PROGRAM F22_AggregationHandScanner
VAR

	fbBarcodeType					: FB_SYSTEM_BarcodeType;

	bPackBarcode					: BOOL;
	bOuterIntermediateBarcode		: BOOL;
	bOuterBarcode					: BOOL;
	bCaseBarcode					: BOOL;
	sPackBarcode					: T_PACK_Barcode;
	sOuterIntermediateBarcode		:  T_MaxString;
	sOuterBarcode					: T_OUTER_Barcode;
	sCaseBarcode					: T_CASE_Barcode;

	fbFindAndDeleteOuter			: FB_CASE_FindAndDeleteOuter;

END_VAR
VAR // added by the converter: edge detectors and wires of the graphical bodies
    _w1, _w2 : BOOL;
END_VAR

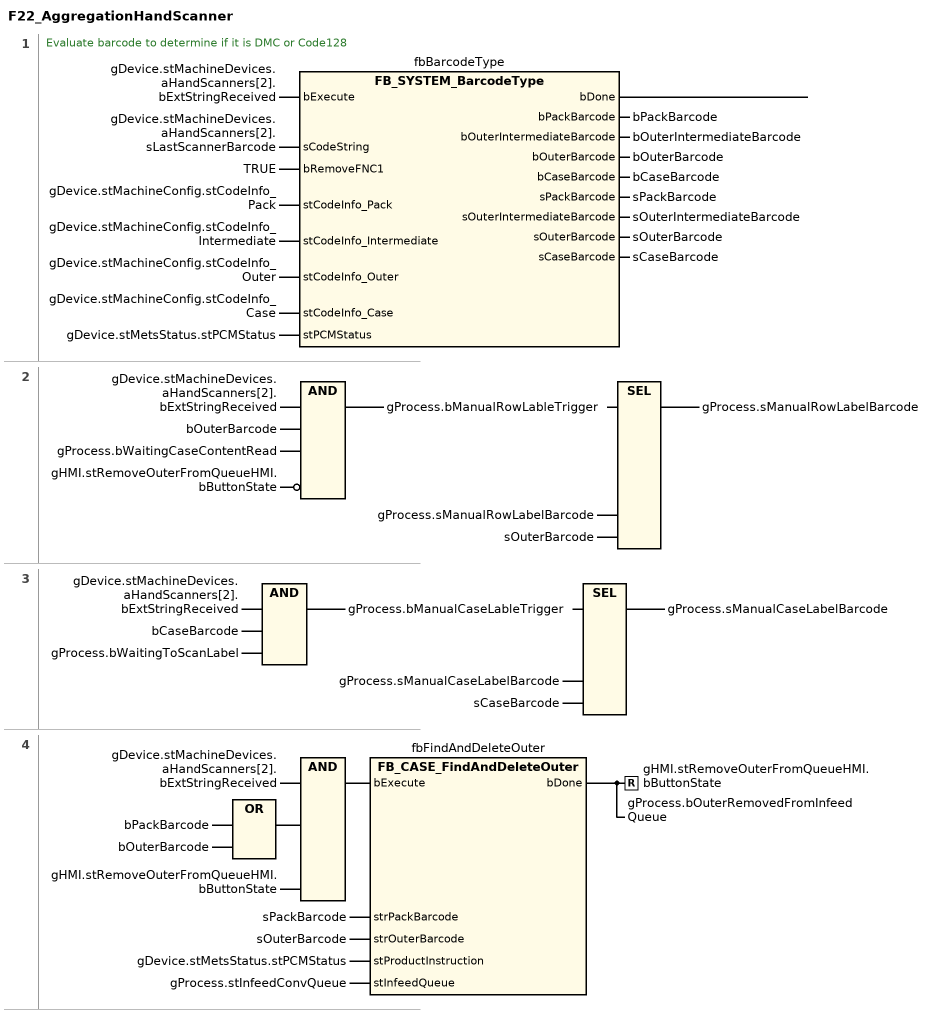
// NETWORK 1
// Evaluate barcode to determine if it is DMC or Code128
fbBarcodeType(
    bExecute := gDevice.stMachineDevices.aHandScanners[2].bExtStringReceived,
    sCodeString := gDevice.stMachineDevices.aHandScanners[2].sLastScannerBarcode,
    bRemoveFNC1 := TRUE,
    stCodeInfo_Pack := gDevice.stMachineConfig.stCodeInfo_Pack,
    stCodeInfo_Intermediate := gDevice.stMachineConfig.stCodeInfo_Intermediate,
    stCodeInfo_Outer := gDevice.stMachineConfig.stCodeInfo_Outer,
    stCodeInfo_Case := gDevice.stMachineConfig.stCodeInfo_Case,
    stPCMStatus := gDevice.stMetsStatus.stPCMStatus,
    bPackBarcode => bPackBarcode,
    bOuterIntermediateBarcode => bOuterIntermediateBarcode,
    bOuterBarcode => bOuterBarcode,
    bCaseBarcode => bCaseBarcode,
    sPackBarcode => sPackBarcode,
    sOuterIntermediateBarcode => sOuterIntermediateBarcode,
    sOuterBarcode => sOuterBarcode,
    sCaseBarcode => sCaseBarcode); // FB_SYSTEM_BarcodeType

// NETWORK 2
_w1 := gDevice.stMachineDevices.aHandScanners[2].bExtStringReceived AND bOuterBarcode AND gProcess.bWaitingCaseContentRead AND NOT gHMI.stRemoveOuterFromQueueHMI.bButtonState;
gProcess.bManualRowLableTrigger := _w1;
gProcess.sManualRowLabelBarcode := SEL(_w1, gProcess.sManualRowLabelBarcode, sOuterBarcode);

// NETWORK 3
_w2 := gDevice.stMachineDevices.aHandScanners[2].bExtStringReceived AND bCaseBarcode AND gProcess.bWaitingToScanLabel;
gProcess.bManualCaseLableTrigger := _w2;
gProcess.sManualCaseLabelBarcode := SEL(_w2, gProcess.sManualCaseLabelBarcode, sCaseBarcode);

// NETWORK 4
fbFindAndDeleteOuter(
    bExecute := gDevice.stMachineDevices.aHandScanners[2].bExtStringReceived AND (bPackBarcode OR bOuterBarcode) AND gHMI.stRemoveOuterFromQueueHMI.bButtonState,
    strPackBarcode := sPackBarcode,
    strOuterBarcode := sOuterBarcode,
    stProductInstruction := gDevice.stMetsStatus.stPCMStatus,
    stInfeedQueue := gProcess.stInfeedConvQueue); // FB_CASE_FindAndDeleteOuter
gHMI.stRemoveOuterFromQueueHMI.bButtonState R= fbFindAndDeleteOuter.bDone;
gProcess.bOuterRemovedFromInfeedQueue := fbFindAndDeleteOuter.bDone;

END_PROGRAM

(* stored: Version 1.1.0.1
   POU F22_AggregationHandScanner: Id {20aaa5bc-60e0-4b8d-b6b0-985dcae6f104}, SpecialFunc None *)
